# EPICS autosave request: stdApp/Db/swait_settings.req
# FILE... swait_settings.req
# USAGE.. swait Record fields autosave'd.
$(P).DESC
$(P).INAN
$(P).INBN
$(P).INCN
$(P).INDN
$(P).INEN
$(P).INFN
$(P).INGN
$(P).INHN
$(P).ININ
$(P).INJN
$(P).INKN
$(P).INLN
$(P).INAP
$(P).INBP
$(P).INCP
$(P).INDP
$(P).INEP
$(P).INFP
$(P).INGP
$(P).INHP
$(P).INIP
$(P).INJP
$(P).INKP
$(P).INLP
$(P).CALC
$(P).OUTN
$(P).OOPT
$(P).DOPT
$(P).DOLN
$(P).SCAN
$(P).ODLY
$(P).PREC
$(P).OEVT
